{attribute 'qualified_only'}
{attribute 'strict'}
TYPE E_SAFETYDOOR :
(
	IDLE := 0,
	SAFETY,
	UNLOCKING,
	UNLOCKED,
	LOCKED,
	WAIT_LOCKED,
	WAIT_UNLOCKED,
	REQUEST_LOCK,
	WAIT_ROBOT
);
END_TYPE

(* stored: Version 1.1.0.1, ProductVersion 3.1.4024.12
   DUT E_SAFETYDOOR: Id {5b3f7e85-5778-4f82-bc9f-18824c990806} *)
